// TIA Portal project "lab7" (V15)

(* hardware
DEVICE "S7-1200 station_1"  S7-1200 Station
   slot 0: "Rack_0"  S7-1200 Rack  Rack  V1.0
   slot 1: "PLC_1"  CPU 1214C DC/DC/DC  6ES7 214-1AG40-0XB0  V4.2
      slot 3: "AQ 1x12BIT_1"  AQ1 signal board  6ES7 232-4HA30-0XB0  V1.0
   slot 101: "CM 1243-5"  CM 1243-5  6GK7 243-5DX30-0XE0  V1.3
   slot 102: "CM 1241 (RS485)_1"  CM 1241 (RS485)  6ES7 241-1CH30-0XB0  V1.0
*)

// ===== PLC "PLC_1"  CPU 1214C DC/DC/DC =====

VAR_GLOBAL   // PLC tag table "Default tag table"
   "start1" AT %I0.0 : Bool;
   "sprzez" AT %M0.0 : Bool;
   "Tag_1" AT %MB10 : Byte;
   "Tag_2" AT %MB12 : Byte;
   "Kierunek" AT %I0.1 : Bool;
   "Tag_4" AT %QB0 : Byte;
END_VAR

// folder: System blocks/Program resources

DATA_BLOCK "t1"   // DB1
{ S7_Optimized_Access := 'TRUE' }
AUTHOR : Simatic
FAMILY : IEC
NAME : IEC_TMR
VERSION : 1.0
// stored: InstanceOfName IEC_TIMER
"IEC_TIMER"
BEGIN
END_DATA_BLOCK

// folder: (top level)

ORGANIZATION_BLOCK "Main"   // OB1, LAD, ProgramCycle
TITLE = "Main Program Sweep (Cycle)"
{ S7_Optimized_Access := 'TRUE' }
VERSION : 0.1
   VAR_INPUT
      Initial_Call : Bool;   // Initial call of this OB
      Remanence : Bool;   // =True, if remanent data are available
   END_VAR
BEGIN

REGION Network 1: generator szpilkowy
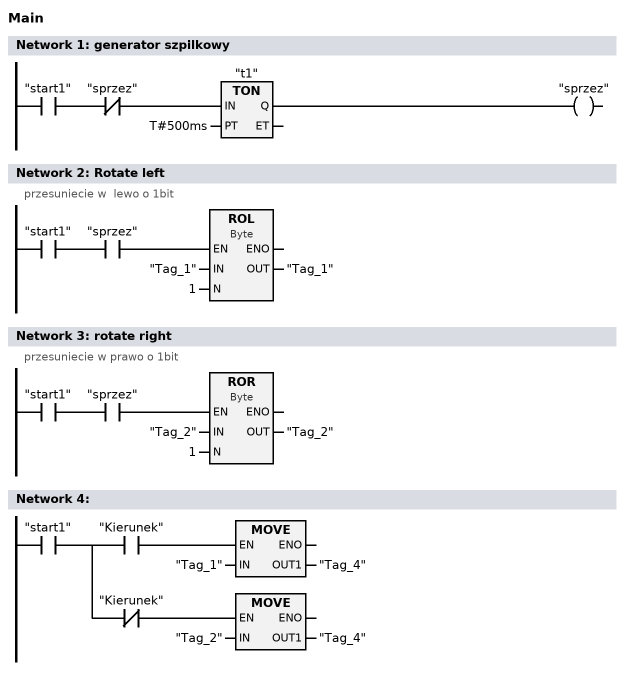
   "t1".TON(IN := "start1" AND NOT "sprzez", PT := T#500ms);
   "sprzez" := "t1".Q;
END_REGION

REGION Network 2: Rotate left
   // przesuniecie w  lewo o 1bit
   IF "start1" AND "sprzez" THEN "Tag_1" := ROL(IN := "Tag_1", N := 1); END_IF;
END_REGION

REGION Network 3: rotate right
   // przesuniecie w prawo o 1bit
   IF "start1" AND "sprzez" THEN "Tag_2" := ROR(IN := "Tag_2", N := 1); END_IF;
END_REGION

REGION Network 4
   RUNG wire#powerrail
      Contact( "start1" )
      wire#w1
      Contact( "Kierunek" )
      Move(in := "Tag_1", out1 => "Tag_4")
   END_RUNG
   RUNG wire#w1
      I_Contact( "Kierunek" )
      Move(in := "Tag_2", out1 => "Tag_4")
   END_RUNG
   // the same network as SCL:
   IF "start1" AND "Kierunek" THEN "Tag_4" := "Tag_1"; END_IF;
   IF "start1" AND NOT "Kierunek" THEN "Tag_4" := "Tag_2"; END_IF;
END_REGION
END_ORGANIZATION_BLOCK

ORGANIZATION_BLOCK "Startup"   // OB100, LAD, Startup
TITLE = "Complete Restart"
{ S7_Optimized_Access := 'TRUE' }
VERSION : 0.1
// blok wywoływany tylko raz przy starcie
   VAR_INPUT
      LostRetentive : Bool;   // True if retentive data are lost
      LostRTC : Bool;   // True if date and time are lost
   END_VAR
BEGIN

REGION Network 1
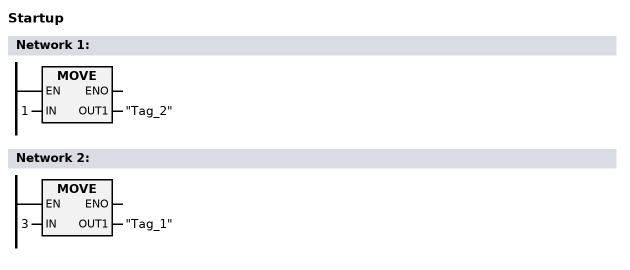
   RUNG wire#powerrail
      Move(in := 1, out1 => "Tag_2")
   END_RUNG
   // the same network as SCL:
   "Tag_2" := 1;
END_REGION

REGION Network 2
   RUNG wire#powerrail
      Move(in := 3, out1 => "Tag_1")
   END_RUNG
   // the same network as SCL:
   "Tag_1" := 3;
END_REGION
END_ORGANIZATION_BLOCK